// SIMATIC S7-200 project (STEP 7-Micro/WIN), CPU 224 REL 02.01

SYMBOL_TABLE 用户定义1
hight            VW401
END_SYMBOL_TABLE

ORGANIZATION_BLOCK 主程序:OB1
TITLE=程序注释  本程序是用库的mbus协议，要安装了库才能使用的
BEGIN
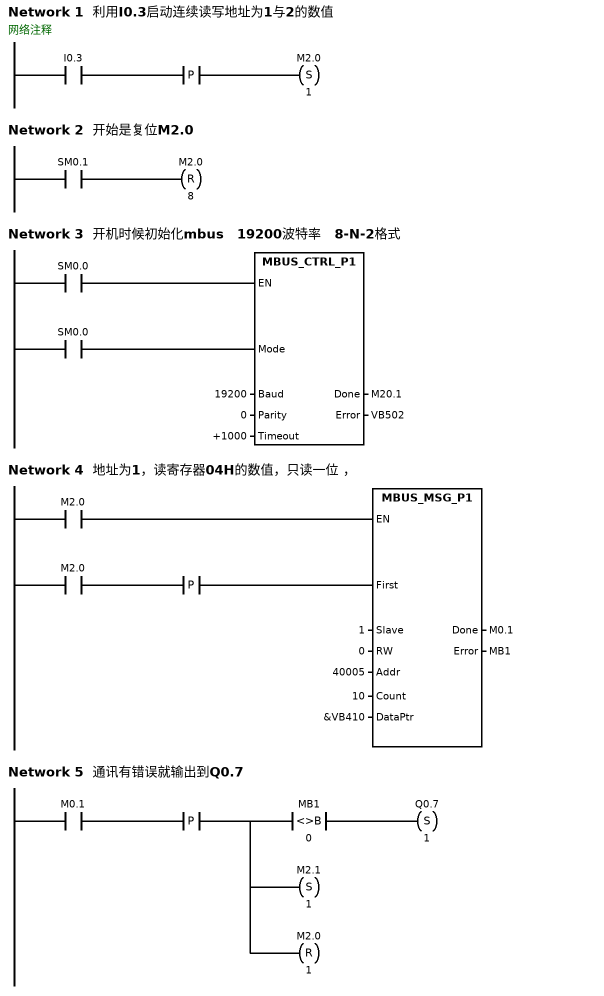
Network 1 // 利用I0.3启动连续读写地址为1与2的数值
// 网络注释
LD     I0.3
EU
S      M2.0, 1
Network 2 // 开始是复位M2.0
LD     SM0.1
R      M2.0, 8
Network 3 // 开机时候初始化mbus   19200波特率   8-N-2格式  
LD     SM0.0
=      L60.0
LD     SM0.0
=      L63.7
LD     L60.0
CALL   MBUS_CTRL_P1:SBR1, L63.7, 19200, 0, +1000, M20.1, VB502
Network 4 // 地址为1，读寄存器04H的数值，只读一位 ，
LD     M2.0
=      L60.0
LD     M2.0
EU
=      L63.7
LD     L60.0
CALL   MBUS_MSG_P1:SBR2, L63.7, 1, 0, 40005, 10, &VB410, M0.1, MB1
Network 5 // 通讯有错误就输出到Q0.7
LD     M0.1
EU
LPS
AB<>   MB1, 0
S      Q0.7, 1
LRD
S      M2.1, 1
LPP
R      M2.0, 1
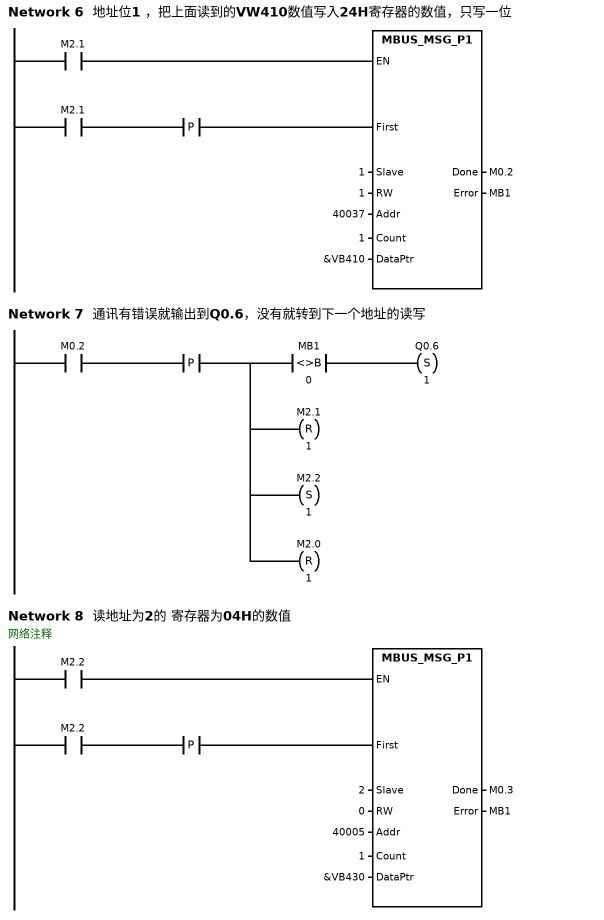
Network 6 // 地址位1 ，把上面读到的VW410数值写入24H寄存器的数值，只写一位
LD     M2.1
=      L60.0
LD     M2.1
EU
=      L63.7
LD     L60.0
CALL   MBUS_MSG_P1:SBR2, L63.7, 1, 1, 40037, 1, &VB410, M0.2, MB1
Network 7 // 通讯有错误就输出到Q0.6，没有就转到下一个地址的读写
LD     M0.2
EU
LPS
AB<>   MB1, 0
S      Q0.6, 1
LRD
R      M2.1, 1
LRD
S      M2.2, 1
LPP
R      M2.0, 1
Network 8 // 读地址为2的 寄存器为04H的数值
// 网络注释
LD     M2.2
=      L60.0
LD     M2.2
EU
=      L63.7
LD     L60.0
CALL   MBUS_MSG_P1:SBR2, L63.7, 2, 0, 40005, 1, &VB430, M0.3, MB1
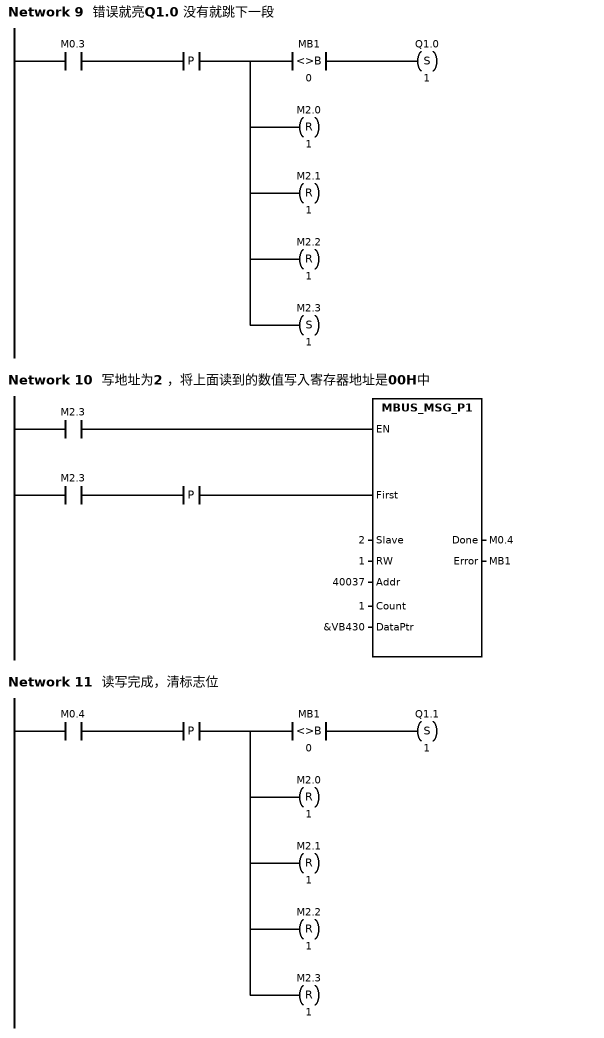
Network 9 // 错误就亮Q1.0 没有就跳下一段
LD     M0.3
EU
LPS
AB<>   MB1, 0
S      Q1.0, 1
LRD
R      M2.0, 1
LRD
R      M2.1, 1
LRD
R      M2.2, 1
LPP
S      M2.3, 1
Network 10 // 写地址为2 ，将上面读到的数值写入寄存器地址是00H中
LD     M2.3
=      L60.0
LD     M2.3
EU
=      L63.7
LD     L60.0
CALL   MBUS_MSG_P1:SBR2, L63.7, 2, 1, 40037, 1, &VB430, M0.4, MB1
Network 11 // 读写完成，清标志位
LD     M0.4
EU
LPS
AB<>   MB1, 0
S      Q1.1, 1
LRD
R      M2.0, 1
LRD
R      M2.1, 1
LRD
R      M2.2, 1
LPP
R      M2.3, 1
END_ORGANIZATION_BLOCK

// SBR1: protected block, not included

// SBR2: protected block, not included

// SBR3: protected block, not included
